(* LS Electric XG5000 project: 05_Practice5_Counter *)
(* PLC LSPLC *)
(* module base 0 slot 0: 입력 모듈:XGI-D21A (DC 24V 입력, 8점 (전류소스/싱크입력)) *)
(* module base 0 slot 1: 출력 모듈:XGQ-RY1A (릴레이 출력, 8점 (2A용, 단독 COM.)) *)

PROGRAM NewProgram (* task: 스캔 프로그램 *)
VAR
    리셋 : BOOL;
    세척밸브 AT %QX0.1.0 : BOOL;
    스위치 AT %IX0.0.0 : BOOL;
    인원카운터 : CTU_INT;
    타이머물공급1 : TP;
    타이머물공급2 : TP;
    타이머물나오기 : TP;
    타이머앉기 : TON;
END_VAR

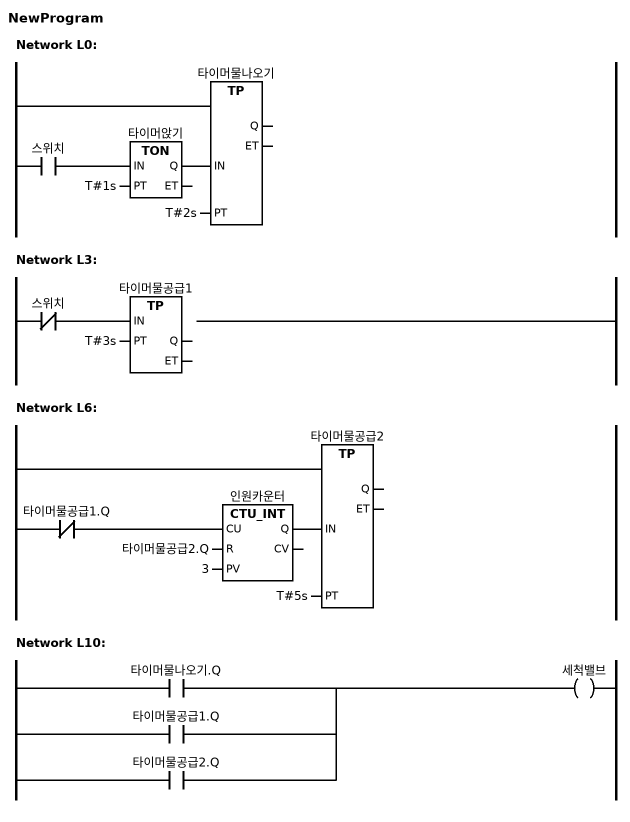
(* Rung L0 *)
타이머앉기(IN := 스위치, PT := T#1s);
타이머물나오기(IN := 타이머앉기.Q, PT := T#2s);
(* Rung L3 *)
타이머물공급1(IN := NOT 스위치, PT := T#3s);
(* Rung L6 *)
인원카운터(CU := NOT 타이머물공급1.Q, R := 타이머물공급2.Q, PV := 3);
타이머물공급2(IN := 인원카운터.Q, PT := T#5s);
(* Rung L10 *)
세척밸브 := 타이머물나오기.Q OR 타이머물공급1.Q OR 타이머물공급2.Q;
END_PROGRAM